FUNCTION_BLOCK Producer
  (* Standard: 61499-2 *)
  (* Version 1.0, 2026-07-29, Dimitrios Kalligaridis *)
  PACKAGE mypackage;
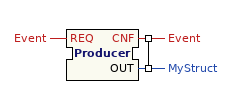
  EVENT_INPUT
    REQ;
  END_EVENT
  EVENT_OUTPUT
    CNF WITH OUT;
  END_EVENT
  VAR_OUTPUT
    OUT : mypackage::MyStruct;
  END_VAR
END_FUNCTION_BLOCK
